// Mitsubishi GX Works2 project: group_18 8.12   PLC: FX3G

// global labels: Global1
VAR_GLOBAL
  Start_day AT X007 : BOOL;
  Working AT Y000 : BOOL;
  End_day AT X005 : BOOL;
  Supply AT M7 : BOOL;
  Input_1 AT D8280 : INT;
  Protein AT D8201 : INT;
  Input_2 AT D8281 : INT;
  Output AT D8282 : INT;
  Oatmeal AT D8202 : INT;
  Honey AT D8203 : INT;
  Mixing AT X003 : BOOL;
END_VAR
VAR_GLOBAL CONSTANT
  number_5 : INT := 1989;
END_VAR
VAR_GLOBAL
  Classic AT M4 : BOOL;
  light2 AT Y002 : BOOL;
END_VAR
VAR_GLOBAL CONSTANT
  number_10 : INT := 4015;
END_VAR
VAR_GLOBAL
  Protein_Snack AT M3 : BOOL;
  Classic_Snack AT M4 : BOOL;
END_VAR
VAR_GLOBAL CONSTANT
  number_400 : INT := 400;
  number_320 : INT := 320;
  number_160 : INT := 160;
END_VAR
VAR_GLOBAL
  timer_5 AT TC5 : BOOL;
END_VAR
VAR_GLOBAL CONSTANT
  number_500 : INT := 2025;
  number_50 : INT := 50;
END_VAR
VAR_GLOBAL
  Mixing_flag AT TS5 : BOOL;
  Mixing_light AT Y003 : BOOL;
END_VAR
VAR_GLOBAL CONSTANT
  number_4 : INT := 4;
  number_240 : INT := 240;
  number_120 : INT := 120;
END_VAR
VAR_GLOBAL
  FinishMix AT M20 : BOOL;
  Baking AT X002 : BOOL;
  Cooking AT M9 : BOOL;
END_VAR
VAR_GLOBAL CONSTANT
  num_5 : INT := 503;
END_VAR
VAR_GLOBAL
  BakeTime AT D8210 : INT;
END_VAR
VAR_GLOBAL CONSTANT
  number_40 : INT := 40;
  num_50 : INT := 50;
END_VAR
VAR_GLOBAL
  BakingTimer AT TC2 : BOOL;
  BakingTimerflag AT TS2 : BOOL;
  BlinkLight AT M11 : BOOL;
  BlinkLight2 AT TC3 : BOOL;
END_VAR
VAR_GLOBAL CONSTANT
  number_20 : INT := 20;
END_VAR
VAR_GLOBAL
  BlinkLight3 AT TC4 : BOOL;
  BlinkLight2Flag AT TS3 : BOOL;
  BlinkLightFlag3 AT TS4 : BOOL;
  Light1 AT Y001 : BOOL;
END_VAR
VAR_GLOBAL CONSTANT
  number_1 : INT := 1;
END_VAR
VAR_GLOBAL
  Flag_True AT M20 : BOOL;
  MixingFlag AT M30 : BOOL;
  Packing AT X006 : BOOL;
  onePiece AT X000 : BOOL;
  packageCounter AT CC0 : BOOL;
END_VAR
VAR_GLOBAL CONSTANT
  number_8 : INT := 8;
END_VAR
VAR_GLOBAL
  BakingStop AT M40 : BOOL;
  CountFinsih AT CS0 : BOOL;
  packageLight AT Y004 : BOOL;
  PackageAmount AT D1200 : INT;
  DuringMix AT M50 : BOOL;
  Starting_Honey AT D1220 : INT;
  Starting_Oatmeal AT D1210 : INT;
  Starting_Protein AT D1230 : INT;
END_VAR

// task Task_01 (event TRUE, interval 0, priority 31): POU_01

PROGRAM POU_01
(* structured ladder/FBD written out as ST: instructions are called as NAME(EN, inputs, outputs); _pN, _eN, _tN stand for wires *)
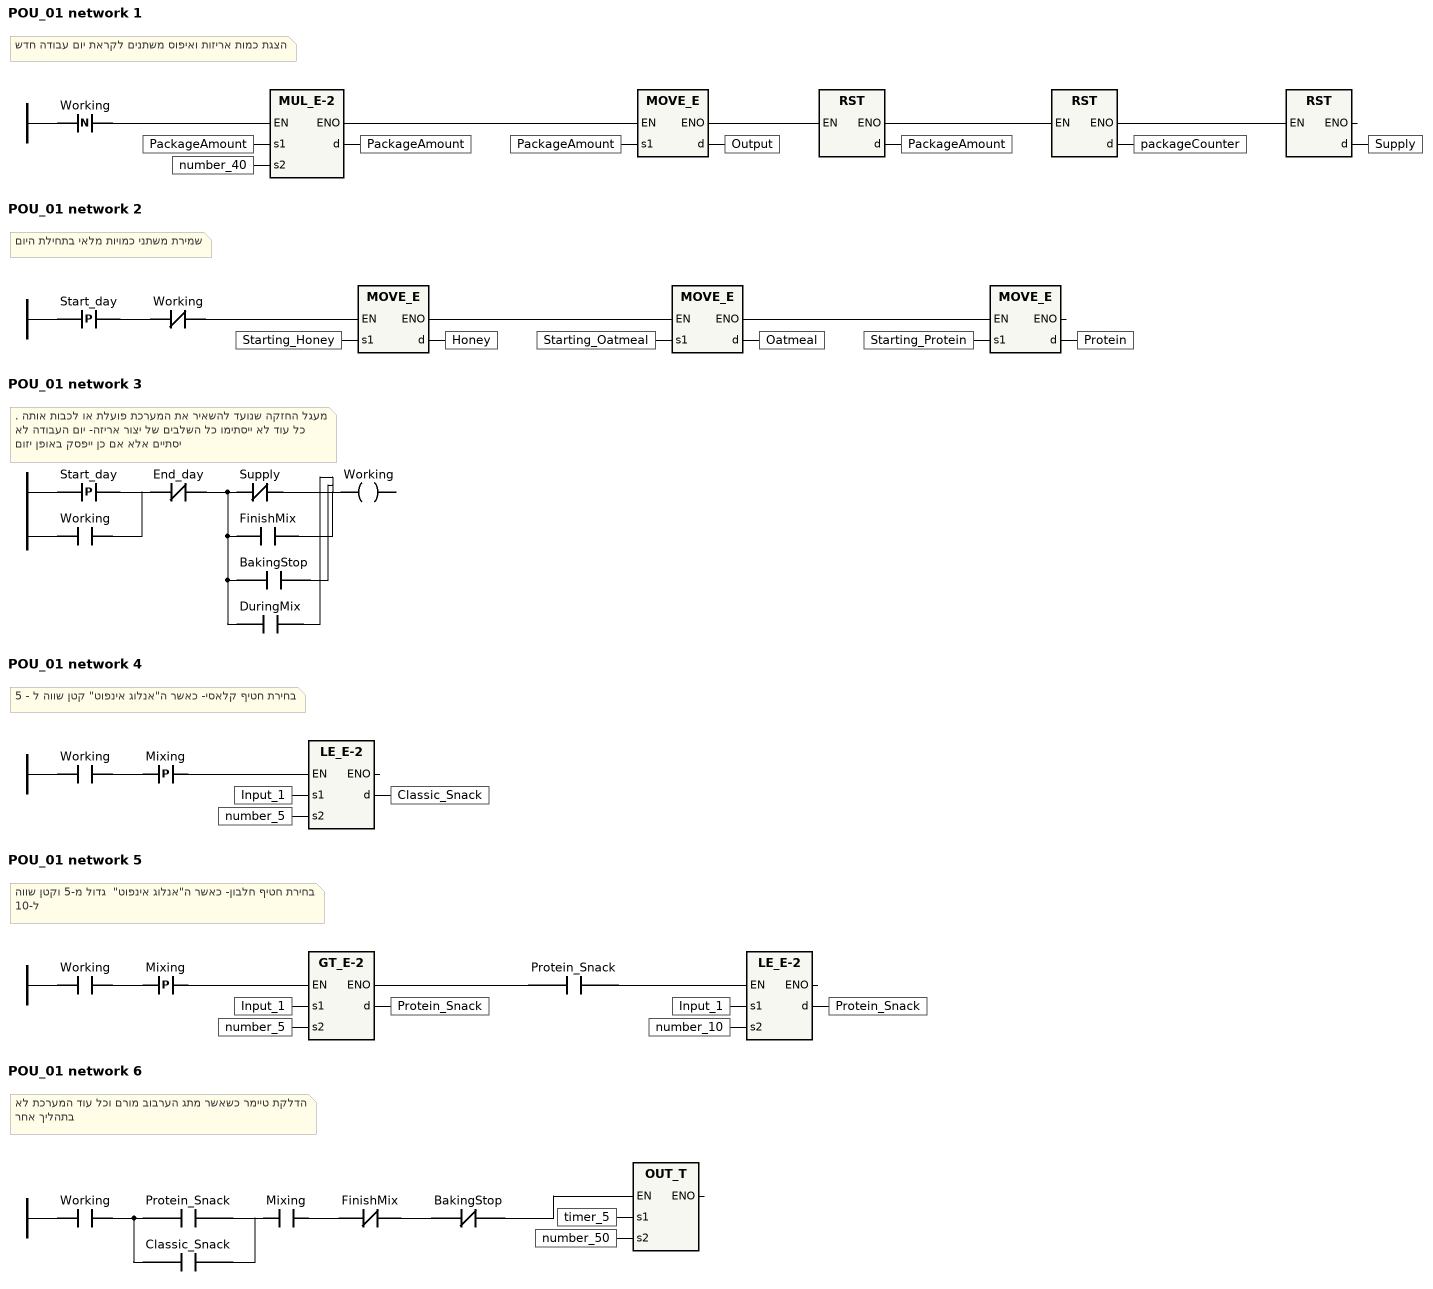
(* network 1 *)
(* הצגת כמות אריזות ואיפוס משתנים לקראת יום עבודה חדש *)
_e1 := MUL_E(LDF(TRUE, Working), PackageAmount, number_40, PackageAmount);
_e2 := MOVE_E(_e1, PackageAmount, Output);
_e3 := RST(_e2, PackageAmount);
_e4 := RST(_e3, packageCounter);
RST(_e4, Supply);
(* network 2 *)
(* שמירת משתני כמויות מלאי בתחילת היום *)
_e1 := MOVE_E(LDP(TRUE, Start_day) AND NOT Working, Starting_Honey, Honey);
_e2 := MOVE_E(_e1, Starting_Oatmeal, Oatmeal);
MOVE_E(_e2, Starting_Protein, Protein);
(* network 3 *)
(* מעגל החזקה שנועד להשאיר את המערכת פועלת או לכבות אותה . כל עוד לא ייסתימו כל השלבים של יצור אריזה- יום העבודה לא יסתיים אלא אם כן ייפסק באופן יזום *)
_p1 := (LDP(TRUE, Start_day) OR Working) AND NOT End_day;
Working := (_p1 AND NOT Supply) OR (_p1 AND FinishMix) OR (_p1 AND BakingStop) OR (_p1 AND DuringMix);
(* network 4 *)
(* בחירת חטיף קלאסי- כאשר ה"אנלוג אינפוט" קטן שווה ל - 5 *)
LE_E(Working AND LDP(TRUE, Mixing), Input_1, number_5, Classic_Snack);
(* network 5 *)
(* בחירת חטיף חלבון- כאשר ה"אנלוג אינפוט"  גדול מ-5 וקטן שווה ל-10 *)
_e1 := GT_E(Working AND LDP(TRUE, Mixing), Input_1, number_5, Protein_Snack);
LE_E(_e1 AND Protein_Snack, Input_1, number_10, Protein_Snack);
(* network 6 *)
(* הדלקת טיימר כשאשר מתג הערבוב מורם וכל עוד המערכת לא בתהליך אחר *)
OUT_T(((((Working AND Protein_Snack) OR (Working AND Classic_Snack)) AND Mixing) AND NOT FinishMix) AND NOT BakingStop, timer_5, number_50);
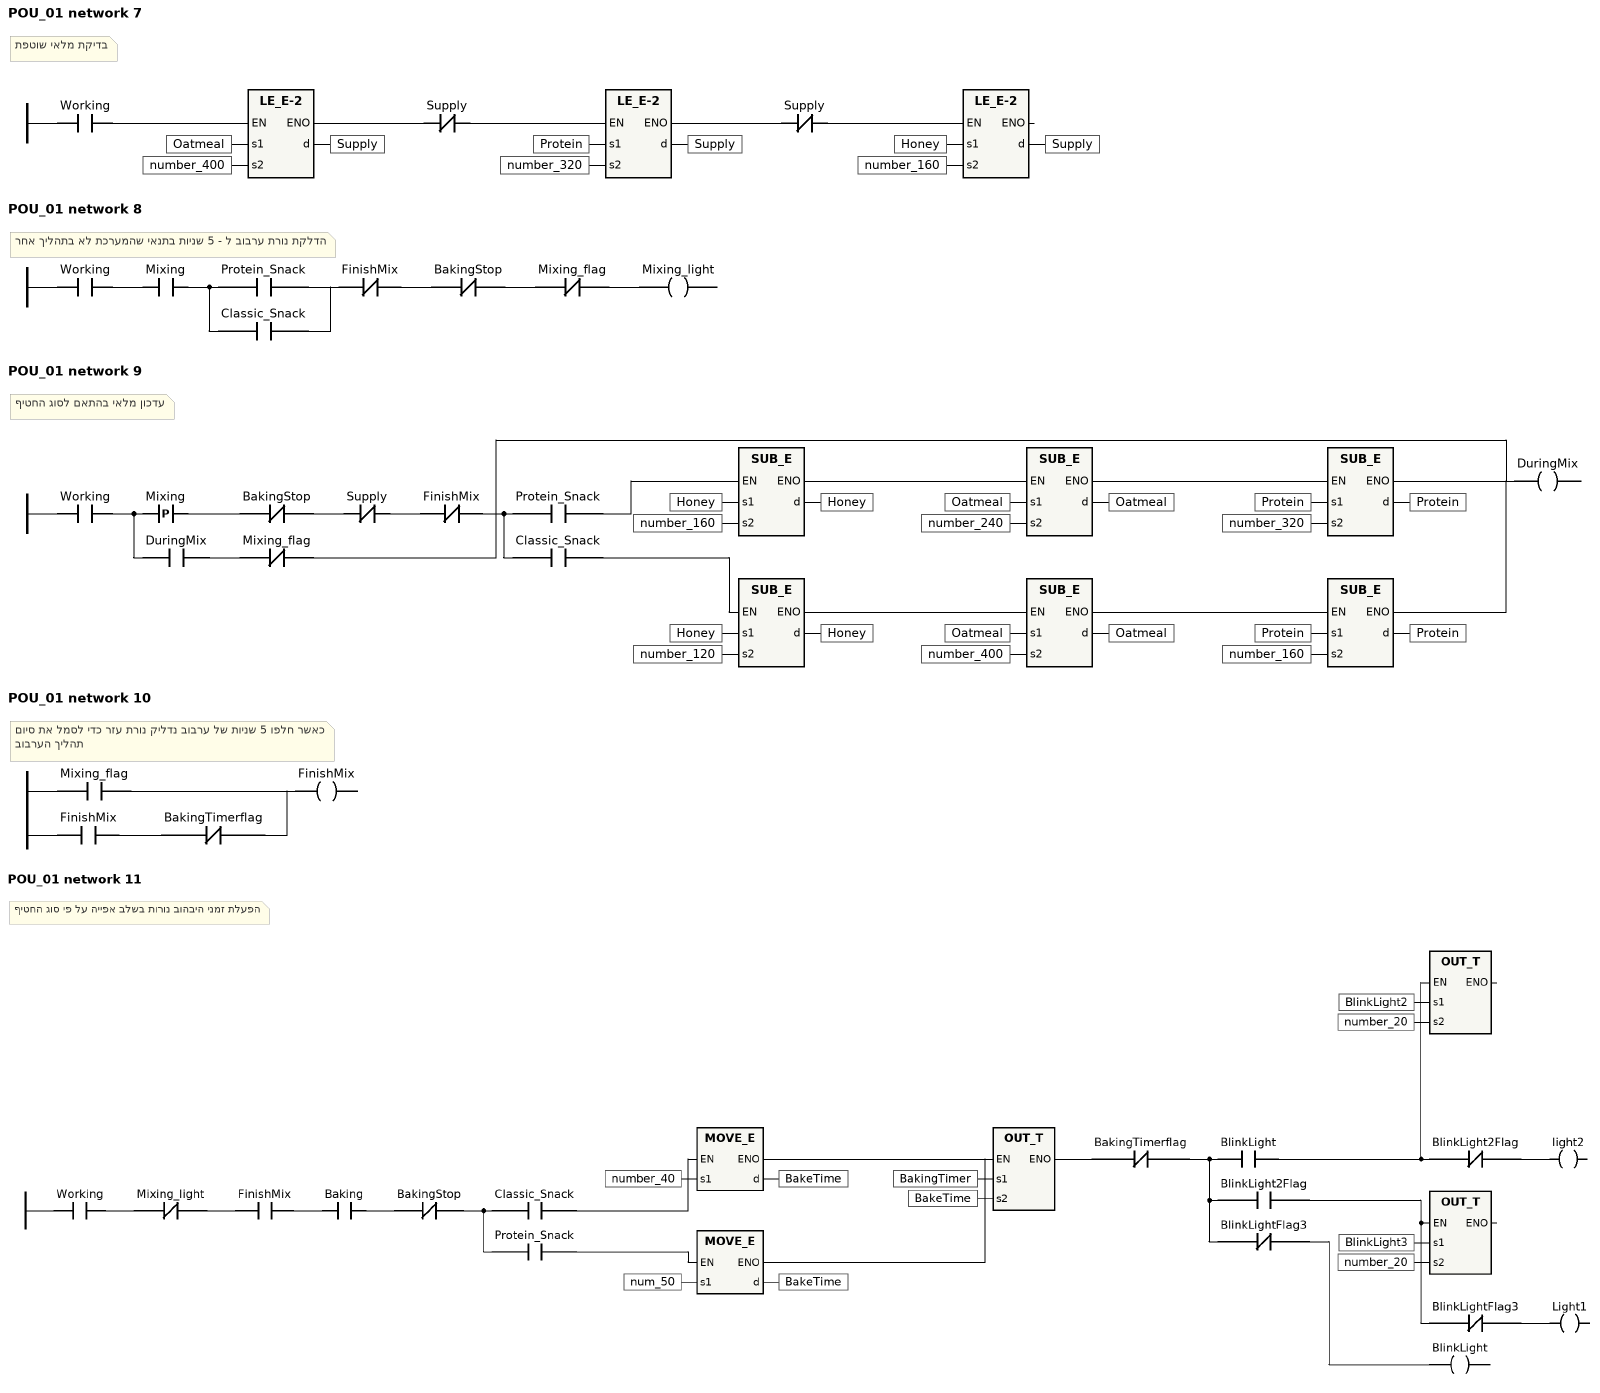
(* network 7 *)
(* בדיקת מלאי שוטפת *)
_e1 := LE_E(Working, Oatmeal, number_400, Supply);
_e2 := LE_E(_e1 AND NOT Supply, Protein, number_320, Supply);
LE_E(_e2 AND NOT Supply, Honey, number_160, Supply);
(* network 8 *)
(* הדלקת נורת ערבוב ל - 5 שניות בתנאי שהמערכת לא בתהליך אחר *)
_p1 := Working AND Mixing;
Mixing_light := ((((_p1 AND Protein_Snack) OR (_p1 AND Classic_Snack)) AND NOT FinishMix) AND NOT BakingStop) AND NOT Mixing_flag;
(* network 9 *)
(* עדכון מלאי בהתאם לסוג החטיף *)
_p1 := Working AND LDP(TRUE, Mixing) AND NOT BakingStop AND NOT Supply AND NOT FinishMix;
_e2 := SUB_E(_p1 AND Protein_Snack, Honey, number_160, Honey);
_e3 := SUB_E(_e2, Oatmeal, number_240, Oatmeal);
_e4 := SUB_E(_e3, Protein, number_320, Protein);
_e5 := SUB_E(_p1 AND Classic_Snack, Honey, number_120, Honey);
_e6 := SUB_E(_e5, Oatmeal, number_400, Oatmeal);
_e7 := SUB_E(_e6, Protein, number_160, Protein);
DuringMix := _e4 OR _e7 OR (Working AND DuringMix AND NOT Mixing_flag);
(* network 10 *)
(* כאשר חלפו 5 שניות של ערבוב נדליק נורת עזר כדי לסמל את סיום תהליך הערבוב *)
FinishMix := Mixing_flag OR (FinishMix AND NOT BakingTimerflag);
(* network 11 *)
(* הפעלת זמני היבהוב נורות בשלב אפייה על פי סוג החטיף *)
_p1 := Working AND NOT Mixing_light AND FinishMix AND Baking AND NOT BakingStop;
_e2 := MOVE_E(_p1 AND Classic_Snack, number_40, BakeTime);
_e3 := MOVE_E(_p1 AND Protein_Snack, num_50, BakeTime);
_e4 := OUT_T(_e2 OR _e3, BakingTimer, BakeTime);
_p5 := _e4 AND NOT BakingTimerflag;
_p6 := _p5 AND BlinkLight;
OUT_T(_p6, BlinkLight2, number_20);
light2 := _p6 AND NOT BlinkLight2Flag;
_p7 := _p5 AND BlinkLight2Flag;
OUT_T(_p7, BlinkLight3, number_20);
Light1 := _p7 AND NOT BlinkLightFlag3;
BlinkLight := _p5 AND NOT BlinkLightFlag3;
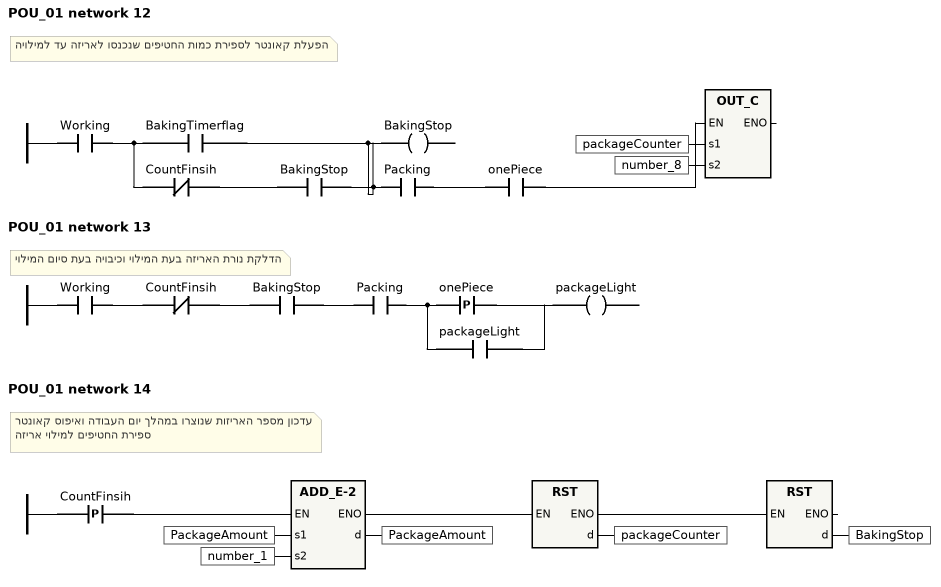
(* network 12 *)
(* הפעלת קאונטר לספירת כמות החטיפים שנכנסו לאריזה עד למילויה *)
_p1 := (Working AND BakingTimerflag) OR (Working AND NOT CountFinsih AND BakingStop);
BakingStop := _p1;
OUT_C(_p1 AND Packing AND onePiece, packageCounter, number_8);
(* network 13 *)
(* הדלקת נורת האריזה בעת המילוי וכיבויה בעת סיום המילוי *)
_p1 := Working AND NOT CountFinsih AND BakingStop AND Packing;
packageLight := (_p1 AND LDP(TRUE, onePiece)) OR (_p1 AND packageLight);
(* network 14 *)
(* עדכון מספר האריזות שנוצרו במהלך יום העבודה ואיפוס קאונטר ספירת החטיפים למילוי אריזה *)
_e1 := ADD_E(LDP(TRUE, CountFinsih), PackageAmount, number_1, PackageAmount);
_e2 := RST(_e1, packageCounter);
RST(_e2, BakingStop);
END_PROGRAM
